(*********************************** G.D S.p.A. - Technical Department ***********************************
============= PROGRAM INFO ============
FOLDER:             TBD
MACHINES INVOLVED:  TBD 

============= DESCRIPTION =============
csp machine declaration

============= REVISIONS ===============
Date		Version	 	Author      	Description             
----------	-------		------------  	--------------------------------------------
2019/04/05 	0000.00	 	M.Grasso		Creation of the PRG

**********************************************************************************************************)
(*$R process_ref := prc; $*)
PROGRAM csp_transfer_infeed_accumulation_level_low
VAR
	
	
	prc:											process;
	prc_path:										STRING;
	
	di_flt:											filter;
	di_status:										BOOL;
	di_presence:									BOOL; (*$M $*)
	di_accumulation:								BOOL;
	
	min_flt_timer_off_on:							DINT:= 2000; (*$P min := 0; max := 10000; step := 1; unit :=  ms; desc := Timer OFF to ON; $*)
	min_flt_timer_on_off:							DINT:= 1000; (*$P min := 0; max := 10000; step := 1; unit :=  ms; desc := Timer ON to OFF; $*)

	
END_VAR

VAR_INPUT
	di:												digital_input;
END_VAR

_read_var_input();

_object_manager();

IF NOT objects_running()
THEN
	RETURN;	
END_IF

_read_process_image();

_mode_manager();

CASE process_get_mode(prc) OF
	MODE_ABSENT,
	MODE_INACTIVE:
		RETURN;
	MODE_TEST:
		_handle_process_test();
END_CASE


_set_runtime_properties();

(********************************* BODY *********************************)
(************************************************************************)

di_status := digital_input_is_active(di);

filter_set_delays(
	delay_off_on := csp_transfer_infeed_accumulation_level.one_carton_in_ms,
	delay_on_off := csp_transfer_infeed_accumulation_level.one_carton_in_ms,
	CONVERSION_this := di_flt);

IF di_status = TRUE
THEN 
	di_presence := TRUE;
	IF filter_is_on(di_flt) 
	THEN
		di_accumulation := TRUE;
	END_IF
ELSE 
	di_accumulation := FALSE;
	IF filter_is_off(di_flt) (*di OFF for a time = 5000ms*)
	THEN
		di_presence := FALSE;
	END_IF
END_IF


(************************************************************************)

_handle_messages();

_write_output();

ACTION _handle_messages:
;
END_ACTION

ACTION _handle_process_test:
;
END_ACTION

ACTION _mode_manager:
IF process_mode_req_is_pending(prc)
THEN
    process_apply_mode_req_first_step(prc);
    CASE process_get_mode(prc) OF
        MODE_TO_ABSENT:
			;
        MODE_TO_INACTIVE:
			;
        MODE_TO_TEST:
			;
        MODE_TO_OPERATIONAL:
			;
    END_CASE
    process_apply_mode_req_second_step(prc);
END_IF
END_ACTION

ACTION _object_manager:
IF objects_initialization()
THEN
	sub_process_init(
		object_name					:= 'csp_transfer_infeed_accumulation_level_low.prc', 
		process						:= csp_transfer_infeed_accumulation_level.prc, 
		CONVERSION_this				:= prc);
		
	prc_path 						:= process_get_path(prc);
	
	(* INPUTS *)
	digital_input_init(
		object_name					:= CONCAT(prc_path, '_di'), 
		polarity_direct				:= TRUE, 
		process						:= prc, 
		CONVERSION_this				:= di);
		
	filter_init(
		object_name 				:= CONCAT(prc_path, '_min_flt'),
		delay_off_on				:= min_flt_timer_off_on,
		delay_on_off 				:= min_flt_timer_on_off,
		process			 			:= prc,
		CONVERSION_this 			:= di_flt);

END_IF

IF objects_running()
THEN
	process_cycle(prc);
	filter_cycle(
				input 			:= di_status,
				CONVERSION_this := di_flt);

END_IF
END_ACTION

ACTION _read_process_image:
;
END_ACTION

ACTION _read_var_input:
;
END_ACTION

ACTION _set_runtime_properties:
;
END_ACTION

ACTION _write_output:
;
END_ACTION

END_PROGRAM

(* stored: Version 1.1.0.1, ProductVersion 3.1.4024.3
   POU csp_transfer_infeed_accumulation_level_low: Id {0c05a8a7-e07c-4f86-bc84-596bbf7edd54}, SpecialFunc None
   Action _handle_messages: Id {8f5f4e57-bc84-4b38-a31d-3cbc4ee9e612}
   Action _handle_process_test: Id {1a6e6a51-2bfd-4df6-901f-65d52bf1aae3}
   Action _mode_manager: Id {9c7e556f-ddee-4684-9bd5-31d9fa5049b2}
   Action _object_manager: Id {096a2cd9-1bc6-45c2-9afa-eb175794de99}
   Action _read_process_image: Id {88a2c20e-82cd-4937-a63c-87c716e9324a}
   Action _read_var_input: Id {d73ab47b-ed86-4177-b133-7af19b03710f}
   Action _set_runtime_properties: Id {d9187cb2-3354-4d2d-9aff-511729b2530c}
   Action _write_output: Id {e8c889f1-0270-47e7-adc5-29634e6dafc6} *)
